{attribute 'pack_mode' := '1'}
TYPE ST_GetPathSegmentVehicleCountDataIn :
STRUCT
	sCellID						: STRING(30);	// 
	sSegmentID					: STRING(30);	// 

END_STRUCT
END_TYPE

(* stored: Version 1.1.0.1, ProductVersion 3.1.4024.5
   DUT ST_GetPathSegmentVehicleCountDataIn: Id {57a31351-1fcc-4a67-8ff8-533b81a1a665} *)
